{attribute 'qualified_only'}
VAR_GLOBAL
	OP1_A100 AT %I*: BOOL; 
END_VAR

(* stored: Version 1.1.0.1, ProductVersion 3.1.4024.11
   GVL IO: Id {2085dfde-1e58-43fb-a31d-fc6934733c39} *)
